{attribute 'qualified_only'}
{attribute 'strict'}
TYPE cTraySize :
(
	
	NoSize := 0,
	Small:= 1,
	Large := 2
	
) DINT;
END_TYPE

(* stored: Version 1.1.0.1, ProductVersion 3.1.4024.6
   DUT cTraySize: Id {09e612f7-5bdb-4984-b963-0a64e05d8824} *)
